RoboDK station: Bewegungsattribute.rdk

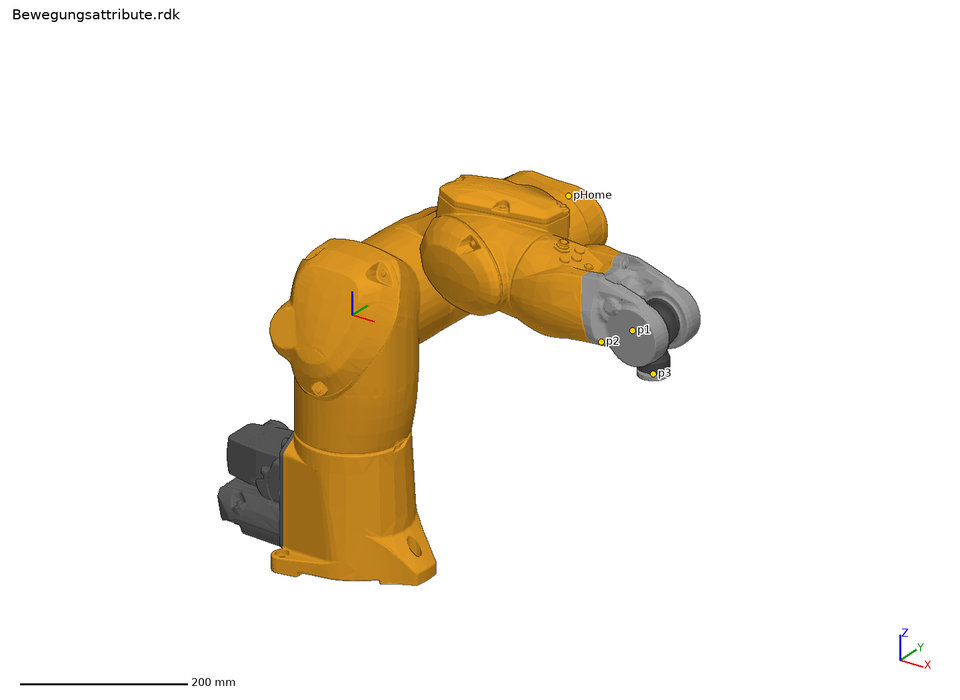
[picture v0: the station drawn from its stored meshes, robots at their saved joint values, targets as dots, program paths as lines]
Station Bewegungsattribute (saved by RoboDK 5.0.2). Poses are relative to the parent item; angles as X-Y-Z fixed-axis rotations.
  - frame Staubli TX2-40 Base at (0, 0, 320) mm
    - robot Staubli TX2-40: 6 axes, payload 1.7 kg, reach 515 mm, repeatability 0.02 mm, weight 29 kg
        modified DH rows (alpha deg, a mm, theta deg, d mm): 0, 0, 0, 320; -90, 0, -90, 35; 0, 225, -90, 0; -90, 0, 0, 225; 90, 0, 0, 0; -90, 0, 180, 65
        base shift (0, 0, -320) mm
        joint limits [-180, -125, -138, -270, -120, -270] to [180, 125, 138, 270, 133.5, 270]; home [0, 0, 90, 0, 0, 0]; saved at [-1.365, 60.05, 34.368, 0, 85.582, -1.365]
    - target pHome (Cartesian target) at (290, 35, 225) mm, rotated rx 0 ry 90 rz 0 deg; joints [0, 0, 90, 0, 0, 0] of Staubli TX2-40
    - target p1 (Cartesian target) at (380, 40, 70) mm, rotated rx 180 ry 0 rz -180 deg; joints [0.753, 44.255, 52.419, 0, 83.325, 0.753] of Staubli TX2-40
    - target p2 (Cartesian target) at (390, -40, 90) mm, rotated rx 180 ry 0 rz 180 deg; joints [-10.978, 47.352, 41.994, 0, 90.653, -10.978] of Staubli TX2-40
    - target p3 (Cartesian target) at (420, 25, 30) mm, rotated rx 180 ry 0 rz -180 deg; joints [-1.365, 60.05, 34.368, 0, 85.582, -1.365] of Staubli TX2-40
  - Python program Bewegungsattribute (listed below)

--- Python program Bewegungsattribute ---
# BEISPIELPROGRAMM: RTS-LIBRARY: BEWEGUNGSATTRIBUTE SETZEN.
# Führt 4 Bewegungen aus, und ändert dann ein Bewegungsattribut.
# Hat KEINE Auswirkung auf die Simulationsattribute, nur auf das Roboterprogramm.

# Import der Librarys
from robolink import *
from robodk import *
from RTS import *

RDK = Robolink()

# Initialisierung aller Simulationsobjekte
rRobot = RDK.Item('Staubli TX2-40')
pHome = RDK.Item('pHome')
p1 = RDK.Item('p1')
p2 = RDK.Item('p2')
p3 = RDK.Item('p3')

# Erstellen des RTS-Objektes. Falls im Programm kein Greifer genutzt wird, muss auch nicht zwingend einer übergeben werden.
RTS = RTS(RDK,rRobot)

RTS.setMovementParameter(30, 30, 30, 30, 30)

# Führt 5 Bewegungen aus
rRobot.MoveJ(pHome)
rRobot.MoveJ(p1)
rRobot.MoveJ(p2)
rRobot.MoveJ(p3)
rRobot.MoveJ(pHome)

# Setzt die maximale Rotationsgeschwindigkeit des Tools. Hat keine Auswirkung auf die Simulation.
RTS.setRotationalSpeedTool(1000)

# Führt 4 Bewegungen aus
rRobot.MoveJ(p1)
rRobot.MoveJ(p2)
rRobot.MoveJ(p3)
rRobot.MoveJ(pHome)

# Setzt die maximale Lineargeschwindigkeit des Tools. Hat keine Auswirkung auf die Simulation.
RTS.setTranslationalSpeedTool(1000)

# Führt 4 Bewegungen aus
rRobot.MoveJ(p1)
rRobot.MoveJ(p2)
rRobot.MoveJ(p3)
rRobot.MoveJ(pHome)

# Setzt die Lineareschwindigkeit des Roboters in % der Nenngeschwindigkeit. Hat keine Auswirkung auf die Simulation.
RTS.setSpeedPercentageJoints(100)

# Führt 4 Bewegungen aus
rRobot.MoveJ(p1)
rRobot.MoveJ(p2)
rRobot.MoveJ(p3)
rRobot.MoveJ(pHome)

# Setzt die Achsbeschleunigung des Roboters in % der Nennbeschleunigung. Hat keine Auswirkung auf die Simulation.
RTS.setAccelerationPercentageJoints(100)

# Führt 4 Bewegungen aus
rRobot.MoveJ(p1)
rRobot.MoveJ(p2)
rRobot.MoveJ(p3)
rRobot.MoveJ(pHome)

# Setzt die Achsverzögerung des Roboters in % der Nennverzögerung. Hat keine Auswirkung auf die Simulation.
RTS.setDeccelerationPercentageJoints(100)

# Führt 4 Bewegungen aus
rRobot.MoveJ(p1)
rRobot.MoveJ(p2)
rRobot.MoveJ(p3)
rRobot.MoveJ(pHome)
